ABB RobotStudio station: Solution_20200503-175143.rsstn

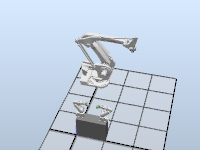
Station Solution (saved by RobotStudio 7.0.8743.626)
Controller Controller, task T_ROB3: task frame (RAPID world) sits at (150, 200, 800) mm in the station
Controller Controller, task T_ROB2: task frame (RAPID world) sits at (150, 200, 800) mm in the station
Controller Controller, task T_ROB1: task frame (RAPID world) sits at (150, 200, 800) mm in the station
Controller Controller
  mechanical unit ROB_1: IRB120_3_58__01, 6 joints, base frame (0, 0, 0) mm
  mechanical unit ROB_2: IRB120_3_58__01_2, 6 joints, base frame (730, 0, 0) mm, rotated rx 0 ry 0 rz 180 deg
  mechanical unit ROB_3: IRB760_450_318__01, 6 joints, base frame (-150, 2800, -800) mm
Layout (positions relative to the parent item):
  - IRB120_3_58__01 [mechanism, from Robots\IRB120_3_58_G_01.rslib] at (150, 200, 800) mm; joint values [0, -0.7064, 0.485, 0, 0.745, 0] (rad or m)
  - IRB120_3_58__01_2 [mechanism, from Robots\IRB120_3_58_G_01.rslib] at (880, 200, 800) mm, rotated rx 0 ry 0 rz 180 deg; joint values [0, -0.8735, 0.5338, 0, 0.8632, 0] (rad or m)
  - IRB760_450_318__01 [mechanism, from Robots\IRB760_450_318__01.rslib] at (0, 3000, 0) mm; joint values [0, -0.5391, -0.1349, 0] (rad or m)
  - Part_1 [part]
  - SimpleGripper [part] at (316.36, 200, 1394) mm, rotated rx 180 ry 60 rz 180 deg
  - SimpleGripper_2 [part] at (763.19, 200, 1394) mm, rotated rx 180 ry 60 rz 0 deg
  - SimpleGripper_3 [part] at (1270.64, 3000, 1824.5) mm, rotated rx 180 ry 0 rz 180 deg
Attachment: SimpleGripper is attached to IRB120_3_58__01 / Link6
Attachment: SimpleGripper_2 is attached to IRB120_3_58__01_2 / Link6
Attachment: SimpleGripper_3 is attached to IRB760_450_318__01 / Link6
